(* IEC 61131-3 sources: Lasal/CPU_5344_V01/Class/cmDrillFeed, 1 file *)

(* ---- cmDrillFeed.st ---- *)
(*!
<Class
	Name               = "cmDrillFeed"
	Revision           = "0.0"
	RealtimeTask       = "false"
	CyclicTask         = "true"
	DefCyclictime      = "10 ms"
	BackgroundTask     = "true"
	DefBackground      = "500 ms"
	Sigmatek           = "false"
	OSInterface        = "false"
	HighPriority       = "false"
	Automatic          = "false"
	UpdateMode         = "Prescan"
	SharedCommandTable = "true"
	Objectsize         = "(480,840)">
	<Channels>
		<Server Name="parPosBack" Visualized="true" Initialize="false" WriteProtected="false" Retentive="SRam"/>
		<Server Name="parTimeBetweenBackAndStop" Visualized="true" Initialize="false" WriteProtected="false" Retentive="SRam"/>
		<Server Name="parTimeBetweenFwdAndBackSkip" Visualized="true" Initialize="false" WriteProtected="false" Retentive="SRam"/>
		<Server Name="parTimeOutTime" Visualized="true" Initialize="false" WriteProtected="false" Retentive="SRam"/>
		<Server Name="stsBeenFwd" Visualized="true" Initialize="false" WriteProtected="true" Retentive="false"/>
		<Server Name="stsPos" Visualized="true" Initialize="false" WriteProtected="false" Retentive="false" Comment="actual position of cilinder"/>
		<Server Name="stsStopBackAtHalf" Visualized="true" Initialize="false" WriteProtected="false" Retentive="false"/>
		<Client Name="iFwdPos" Required="true" Internal="false"/>
		<Client Name="iLivePos" Required="true" Internal="false" Comment="optional actual pos to check with"/>
		<Client Name="iSafeBackPos" Required="true" Internal="false"/>
		<Client Name="iStartFeedPos" Required="true" Internal="false"/>
		<Client Name="iValuesOk" Required="true" Internal="false"/>
		<Client Name="oFeed" Required="true" Internal="false" Comment="optional output for position in"/>
		<Client Name="oSkipValve" Required="true" Internal="false" Comment="optional output for position out"/>
		<Client Name="oStopValve" Required="true" Internal="false"/>
	</Channels>
	<Separators>
		<Servers>
			<SepChn Position="0"/>
			<SepChn Position="4"/>
		</Servers>
	</Separators>
	<Network Name="cmDrillFeed">
		<!-- List of Components in this network -->
		<Components>
			<Object
				Name       = "_base"
				Class      = "cmBase"
				Position   = "(218,120)"
				Visualized = "true">
				<Channels>
					<Server Name="ClassSvr"/>
					<Server Name="cmdHMI"/>
					<Server Name="ErrorNr"/>
					<Server Name="mode"/>
					<Server Name="state"/>
					<Server Name="stsHMI_RunsAllowed"/>
					<Server Name="stsInAlarm"/>
					<Server Name="stsIsInterlocked"/>
					<Client Name="id"/>
					<Client Name="nwEmOrUnit"/>
				</Channels>
			</Object>
		</Components>
		<Comments>
		</Comments>
		<!-- List of Connections in this network -->
		<Connections>
			<Connection Source="this.ClassSvr" Destination="_base.ClassSvr" Vertices="(1036,210),(864,210),"/>
			<Connection Source="this.state" Destination="_base.state" Vertices="(1036,270),(864,270),"/>
			<Connection Source="this.mode" Destination="_base.mode" Vertices="(1036,330),(864,330),"/>
			<Connection Source="this.cmdHMI" Destination="_base.cmdHMI" Vertices="(1036,390),(864,390),"/>
			<Connection Source="this.stsInAlarm" Destination="_base.stsInAlarm" Vertices="(1036,450),(864,510),"/>
			<Connection Source="this.stsIsInterlocked" Destination="_base.stsIsInterlocked" Vertices="(1036,510),(864,570),"/>
			<Connection Source="_base.nwEmOrUnit" Destination="this.nwEmOrUnit" Vertices="(218,210),(38,210),"/>
			<Connection Source="_base.id" Destination="this.id" Vertices="(218,270),(38,270),"/>
			<Connection Source="this.stsHMI_RunsAllowed" Destination="_base.stsHMI_RunsAllowed" Vertices="(1036,570),(864,630),"/>
		</Connections>
		<!-- Headerfiles -->
		<Options>
		</Options>
	</Network>
</Class>
*)
#pragma using cmBase

cmDrillFeed : CLASS
: cmBase
  //Servers:
	stsPos 	: SvrCh_feedPos;
	stsBeenFwd 	: SvrCh_DINT;
	stsStopBackAtHalf 	: SvrCh_DINT;
	parTimeOutTime 	: SvrCh_UDINT;
	parTimeBetweenFwdAndBackSkip 	: SvrCh_UDINT;
	parTimeBetweenBackAndStop 	: SvrCh_UDINT;
	parPosBack 	: SvrCh_DINT;
  //Clients:
	oFeed 	: CltCh_DINT;
	oSkipValve 	: CltCh_DINT;
	oStopValve 	: CltCh_DINT;
	iLivePos 	: CltCh_DINT;
	iStartFeedPos 	: CltCh_DINT;
	iFwdPos 	: CltCh_DINT;
	iSafeBackPos 	: CltCh_DINT;
	iValuesOk 	: CltCh_DINT;
  //Variables:
		timeOutTimer 	: strTimer;
		timerFwdAndSkip 	: strTimer;
		stopTimer 	: strTimer;
		oldStsPos 	: feedPos;
		oldMode 	: eModePML;
  //Functions:

	FUNCTION VIRTUAL work;

	FUNCTION VIRTUAL execStart;

	FUNCTION VIRTUAL execStop;

	FUNCTION VIRTUAL preScanOverride;

	FUNCTION VIRTUAL postScanOverride;

	FUNCTION startMovement
		VAR_OUTPUT
			ok 	: DINT;
		END_VAR;

	FUNCTION stopMovement;

	FUNCTION GLOBAL csStartMovement
		VAR_INPUT
			goBackHalf 	: DINT;
		END_VAR
		VAR_OUTPUT
			ok 	: DINT;
		END_VAR;

	FUNCTION GLOBAL csStopMovement;
  //Tables:
	FUNCTION @STD
		VAR_OUTPUT
			ret_code	: CONFSTATES;
		END_VAR;
	FUNCTION GLOBAL TAB @CT_;
END_CLASS;

// JdK 11-6-2019 class drillfeed, created for library icm project 4284 TraffiRoad
// goal is to control a special drill movement, for this movement we have 3 outputs,
// we have a stopvalve, this one has to be active if we move forward,
// there is a feedvalve, this one is active if moving forward, but also if we have to hold the movement before it's complete back
// and there is a skipvalve, this one is active if we move fast forward, and also if we move back

// only possible movements we have are going forward, then go back complete and going forward and go back until certain value
// in manual mode we always go back complete

// during a interlock state is going back to unknown, this means no active outputs, after a certain time unkown state changes to back
// also if mode changes from auto to manual vice versa, stop movement by going to unkown

// alarms:  1: time-out
//          2: moved from complete back
//          3: no valid values during start

FUNCTION VIRTUAL cmDrillFeed::work

  IF pmlCom.sts.isInterlocked= 1 & stsPos<> fdUnKnown & stsPos<> fdCompleteBack THEN
    stsPos:= fdUnKnown;
  END_IF;
  IF ((pmlCom.sts.mode = auto & (oldMode = manual | oldMode = halfAuto)) | //stop movement if mode changes
      ((pmlCom.sts.mode = manual | pmlCom.sts.mode = halfAuto) & oldMode = auto)) & (stsPos<> fdUnKnown & stsPos<> fdCompleteBack) THEN
    stsPos:= fdUnKnown;
  END_IF;

  oldMode:= pmlCom.sts.mode;

  CASE stsPos OF

  fdUnKnown: //just wait for command, change to complete back if position tells we are complete back
    IF iLivePos >= parPosBack THEN
      stsPos:=fdCompleteBack;
    END_IF;

  fdCompleteBack: //just wait for command, change to unkown if position tells we are not complete back
    IF iLivePos < parPosBack THEN
      giveAlarm(errorNr:=2);
      stsPos:=fdUnKnown;
    END_IF;

  fdMovingFastFwd: //go fast until right pos
    IF iLivePos <= iStartFeedPos THEN
      stsPos:= fdMovingFwd;
    END_IF;
    oFeed:=1;
    oStopValve:=1;
    oSkipValve:=1;

  fdMovingFwd: //go fwd until arrived
    IF iLivePos <= iFwdPos THEN
      stsBeenFwd:= 1;
      stsPos:= fdMovingBack;
    END_IF;
    oFeed:=1;
    oStopValve:=1;

  fdMovingBack: //go back
    IF stsStopBackAtHalf= 1 & iLivePos >= iSafeBackPos THEN
      stsPos:= fdWaitStopBack;
    ELSIF stsStopBackAtHalf= 0 & iLivePos >= parPosBack THEN
      stsPos:= fdCompleteBack;
    END_IF;
    IF timerFwdAndSkip.done= 1 THEN
      oSkipValve:= 1;
    END_IF;

  fdWaitStopBack: //wait some time before we really can stop the movement
    IF stopTimer.done= 1 THEN
      stsPos:= fdStopBack;
    END_IF;

  fdStopBack: //stop in the middle of a movement, in this way the tool is close to the material
    oFeed:=1;
    IF iLivePos >= parPosBack THEN //if state changed in real, also change state in stsPos
      stsPos:=fdCompleteBack;
    END_IF;

  END_CASE;

END_FUNCTION

FUNCTION cmDrillFeed::startMovement
	VAR_OUTPUT
		ok 	: DINT;
	END_VAR

  ok:=0;
  IF stsPos= fdStopBack & iLivePos < iStartFeedPos THEN //tool already close to material, start moving fwd slow
    stsBeenFwd:= 0;
    stsPos:= fdMovingFwd;
    ok:=1;
  ELSIF stsPos= fdCompleteBack | (stsPos= fdStopBack & iLivePos >= iStartFeedPos) THEN //only possible to start movement if drill at stop back, or at complete back
    stsBeenFwd:= 0;
    stsPos:= fdMovingFastFwd;
    ok:=1;
  END_IF;

END_FUNCTION

FUNCTION cmDrillFeed::stopMovement

  IF stsPos <> fdCompleteBack & stsPos <> fdUnKnown THEN
    stsStopBackAtHalf:=0;
    stsPos:=fdMovingBack;
  END_IF;

END_FUNCTION

FUNCTION VIRTUAL cmDrillFeed::execStart

  IF (pmlCom.sts.mode= manual | pmlCom.sts.mode=service) & iValuesOk=1 THEN
    //JdK 26-7-2019 for test stsStopBackAtHalf:=0; //in manual mode always go back complete
    startMovement();
  ELSIF iValuesOk= 0 THEN
    giveAlarm(errorNr:=3);
  END_IF;

END_FUNCTION

FUNCTION VIRTUAL cmDrillFeed::execStop

  IF pmlCom.sts.mode= manual | pmlCom.sts.mode= service THEN
    stopMovement();
  END_IF;

END_FUNCTION

FUNCTION GLOBAL cmDrillFeed::csStartMovement
	VAR_INPUT
		goBackHalf 	: DINT;
	END_VAR
	VAR_OUTPUT
		ok 	: DINT;
	END_VAR

  ok:=0;
  IF pmlCom.sts.mode=auto | pmlCom.sts.mode=service THEN
    IF (stsPos = fdCompleteBack | stsPos = fdStopBack) & iValuesOk=1 THEN
      stsStopBackAtHalf:=goBackHalf;
      ok:=startMovement();
    ELSIF iValuesOk= 0 THEN
      giveAlarm(errorNr:=3);
    END_IF;
  END_IF;

END_FUNCTION

FUNCTION GLOBAL cmDrillFeed::csStopMovement

  IF pmlCom.sts.mode= auto | pmlCom.sts.mode=service THEN
    stopMovement();
  END_IF;

END_FUNCTION

FUNCTION VIRTUAL cmDrillFeed::preScanOverride
//preScan reads in al values before handling the actions

  //first read in all values
  iValuesOk := iValuesOk.Read();
  IF iValuesOk= 1 & stsPos <> fdMovingFwd & stsPos <> fdMovingFastFwd & stsPos <> fdMovingBack & stsPos <> fdWaitStopBack THEN //only reed in if nog drilling is active
    iStartFeedPos := iStartFeedPos.Read();
    iFwdPos := iFwdPos.Read();
    iSafeBackPos := iSafeBackPos.Read();
  END_IF;

  //then call timers
  timeOutTimer:=runTimer(Active:=(stsPos=oldStsPos & stsPos <> fdUnKnown & stsPos <> fdStopBack & stsPos <> fdCompleteBack),
                                                                           iMem:=timeOutTimer, TimerTime:=parTimeOutTime, Pause:=FALSE);
  stopTimer:=runTimer(Active:=stsPos=fdWaitStopBack, iMem:=stopTimer, TimerTime:=parTimeBetweenBackAndStop, Pause:=FALSE);

  timerFwdAndSkip:=runTimer(Active:=stsPos=fdMovingBack, iMem:=timerFwdAndSkip, TimerTime:=parTimeBetweenFwdAndBackSkip, Pause:=FALSE);

  oldStsPos:=stsPos;

  //every cycle set outputs to 0, set them again if asked
  oFeed:=0;
  oSkipValve:=0;
  oStopValve:=0;

  IF pmlCom.cmd.simulation = allSimu THEN
    CASE stsPos OF

    fdMovingFastFwd:
      iLivePos:=iLivePos-10;

    fdMovingFwd:
      iLivePos:=iLivePos-1;

    fdMovingBack:
      iLivePos:=iLivePos+10;

    END_CASE;

    iLivePos.Write(input:=iLivePos);
  ELSE
    iLivePos:=iLivePos.Read();
  END_IF;

END_FUNCTION

FUNCTION VIRTUAL cmDrillFeed::postScanOverride

  //write outputs
  oFeed.Write(input:=oFeed);
  oSkipValve.Write(input:=oSkipValve);
  oStopValve.Write(input:=oStopValve);

  //check alarmstatus
  IF _Alarm.AlarmActief THEN
    stsInAlarm:=1;
  ELSE
    stsInAlarm:=0;
  END_IF;

END_FUNCTION
